(* PLC project 117_1_V0.5.project, CODESYS CODESYS V3.5 SP17 Patch 3 *)
(* stored: creationDateTime 1970-01-01T00:00:00, modificationDateTime 2026-03-26T18:14:32.4070562 *)

FUNCTION_BLOCK BasicPIDController
  VAR
    _Pv : REAL;
    _Sp : REAL;
    _Kp : REAL;
    _Ki : REAL;
    _Kd : REAL;
    _Ts : TIME;
    _Error : REAL;
    _Output : REAL;
    _MinOut : REAL;
    _MaxOut : REAL;
    _Direction : PID_DIRECTION_UDT;
    _PreviousError : REAL;
    _Proportional : REAL;
    _Integral : REAL;
    _Differential : REAL;
    _Status : PID_STATUS_UDT;
  END_VAR

            //Включение ПИД
IF _Status <> Enabled THEN
	Reset();	//Integral := 0; PreviousError := 0;Output := 0;
	RETURN;
ELSE
//Значение текущей ошибки
_Error			:= xError(); //CASE Direction OF DIRECT:xError := (Sp - Pv) * 1.0; REVERSE:xError := (Sp - Pv) * -1.0; END_CASE
// Пропорционал
_Proportional	:= xProportional();	//xProportional := Kp * Error;
// Интеграл
_Integral		:= xIntegral();	//xIntegral := LIMIT(OutMin, (Integral + Ki * Error * ((TIME_TO_REAL (Ts)) / 1000)), OutMax);
// ДиФФеренциал
_Differential	:= xDifferential(); //xDifferential := Kd * (Error - PreviousError) / ((TIME_TO_REAL (Ts)) / 1000);
//Значение предыдущей ошибки
_PreviousError	:= _Error;
//Выход ПИД
_Output := LIMIT(_MinOut, _Proportional + _Integral + _Differential, _MaxOut);
END_IF




          

METHOD Set_Configuration : BOOL
  VAR_INPUT
    Kp : REAL := 0.1;
    Ki : REAL := 0;
    Kd : REAL := 0;
    Ts : TIME := TIME#100ms;
    MinOut : REAL := 0;
    MaxOut : REAL := 100;
    Direction : PID_DIRECTION_UDT := DIRECT;
  END_VAR
                  _Kp 		 := Kp;		
_Ki 		 := Ki;		
_Kd 		 := Kd;		
_Ts			 := Ts;		
_MinOut		 := MinOut;		
_MaxOut		 := MaxOut;	
_Direction   := Direction;
                
END_METHOD
END_FUNCTION_BLOCK
